{attribute 'qualified_only'}
VAR_GLOBAL
END_VAR

(* stored: Version 1.1.0.1, ProductVersion 3.1.4024.10
   GVL Output: Id {c5e20ba5-1bb4-4e9a-a05d-011647d00902} *)
